FUNCTION_BLOCK SUBSCRIBE_0 (* Event-only Subscriber *)
  (* Standard: 61499-2 *)
  (* Version 0.1, 2001-01-27, JHC, Rockwell Automation, Added no_double_init, reinitialize. *)
  (* Version 0.0, 2000-03-23, JHC, Rockwell Automation, Fixed NULL encoding. *)
  (* Compiler header: package fb.rt.net; *)
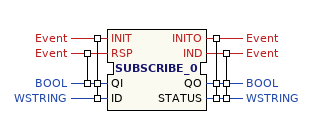
  EVENT_INPUT
    INIT WITH QI, ID; (* Service Initialization *)
    RSP WITH QI; (* Service Response *)
  END_EVENT
  EVENT_OUTPUT
    INITO WITH QO, STATUS; (* Initialization Confirm *)
    IND WITH QO, STATUS; (* Service Indication *)
  END_EVENT
  VAR_INPUT
    QI : BOOL; (* Event Input Qualifier *)
    ID : WSTRING; (* Connection Identifier *)
  END_VAR
  VAR_OUTPUT
    QO : BOOL; (* Event Output Qualifier *)
    STATUS : WSTRING; (* Service Status *)
  END_VAR
  SERVICE SUBSCRIBE_0/Resource (* See PUBLISH_0 for other sequences *)
    SEQUENCE no_double_init
      SUBSCRIBE_0.INIT+(ID) -> Resource.connect(ID) -> SUBSCRIBE_0.INITO+(STATUS);
      SUBSCRIBE_0.INIT+(ID);
    END_SEQUENCE
    SEQUENCE reinitialize
      SUBSCRIBE_0.INIT+(ID) -> Resource.connect(ID) -> SUBSCRIBE_0.INITO+(STATUS);
      SUBSCRIBE_0.INIT-() -> Resource.disconnect() -> SUBSCRIBE_0.INITO-(STATUS);
      SUBSCRIBE_0.INIT+(ID) -> Resource.connect(ID) -> SUBSCRIBE_0.INITO+(STATUS);
    END_SEQUENCE
  END_SERVICE
END_FUNCTION_BLOCK
